// TIA Portal V17 export
// export: Created 2022-07-20T07:01:34.0811229Z, ExportSetting WithDefaults, DisplayName Totally Integrated Automation Portal, DisplayVersion V17, DisplayName TIA Portal Openness, DisplayVersion V17, DisplayName TIA Portal Version Control Interface, DisplayVersion V17, DisplayName SINAMICS Startdrive Advanced, DisplayVersion V17, DisplayName SINAMICS Startdrive G130, G150, S120, S150, SINAMICS MV, S210, DisplayVersion V17, DisplayName SINAMICS Startdrive G110M, G120, G120C, G120D, G120P, G115D, DisplayVersion V17, DisplayName STEP 7 Professional, DisplayVersion V17, DisplayName STEP 7 Safety, DisplayVersion V17, DisplayName WinCC Advanced, DisplayVersion V17
FUNCTION_BLOCK "FB10324_PrinterCompactCapingStation"   // FB10324, LAD
{ S7_Optimized_Access := 'TRUE' }
VERSION : 0.1
// stored: AutoNumber false, IsIECCheckEnabled false, IsRetainMemResEnabled false, MemoryReserve 100, SetENOAutomatically false, UDAEnableTagReadback false
   VAR_OUTPUT
      CapingStation_FillingDone : Bool;
      CapingStationLongOverflowingDone : Bool;
      CapingStationShortOverflowingDone : Bool;
      CapingStationEmptyingDone : Bool;
      CapingStation_WashupSolenoidValve_1_2 : Bool;
      CapingStation_WashupSolenoidValve_3_4 : Bool;
      CapingStation_EmptyingSolenoidValve_1_2 : Bool;
      CapingStation_EmptyingSolenoidValve_3_4 : Bool;
      CapingStation_CleaningSolenoidValve_1_2 : Bool;
      CapingStation_CleaningSolenoidValve_3_4 : Bool;
      CapingStation_WashupPump : Bool;
      CapingStation_EmptyingPump : Bool;
   END_VAR
   VAR_IN_OUT
      RequestFillingCapingStation : Bool;
      RequestLongOverflowingCapingStation : Bool;
      RequestShortOverflowingCapingStation : Bool;
      RequestEmptyingCapingStation : Bool;
   END_VAR
   VAR
      ManagerCapingStationStateDiagram : Int;
      TON_FillingCapingStation : TON_TIME;
      TON_LongOverflowingCapingStation : TON_TIME;
      TON_ShortOverflowingCapingStation : TON_TIME;
      TON_EmptyingCapingStation : TON_TIME;
      R_TRIG_RequestFillingCapingStation { S7_SetPoint := 'True'} : R_TRIG;
      R_TRIG_RequestLongOverflowingCapingStation { S7_SetPoint := 'True'} : R_TRIG;
      R_TRIG_RequestShortOverflowingCapingStation { S7_SetPoint := 'True'} : R_TRIG;
      R_TRIG_RequestEmptyingCapingStation { S7_SetPoint := 'True'} : R_TRIG;
   END_VAR
   VAR CONSTANT
      "0_WAIT_FOR_REQUEST_CAPING_STATION" : Int;
      "10_REQUEST_FILING_CAPING_STATION" : Int := 10;
      "20_REQUEST_LONG_OVERFLOWING_CAPING_STATION" : Int := 20;
      "30_REQUEST_SHORT_OVERFLOWING_CAPING_STATION" : Int := 30;
      "40_REQUEST_EMPTYING_CAPING_STATION" : Int := 40;
      "10000_ALL_ACTIONS_DONE" : Int := 10000;
   END_VAR
BEGIN

REGION Network 1 (SCL): FirstScan
   IF "FirstScan" THEN
       ;
   END_IF;
END_REGION

REGION Network 2 (SCL): Edge Signals & Timers
   REGION EDGE SIGNAL

       #R_TRIG_RequestFillingCapingStation(CLK := #RequestFillingCapingStation);
       #R_TRIG_RequestLongOverflowingCapingStation(CLK := #RequestLongOverflowingCapingStation);
       #R_TRIG_RequestShortOverflowingCapingStation(CLK := #RequestShortOverflowingCapingStation);
       #R_TRIG_RequestEmptyingCapingStation(CLK := #RequestEmptyingCapingStation);

   END_REGION

   REGION

       #TON_FillingCapingStation(IN := #ManagerCapingStationStateDiagram = #"10_REQUEST_FILING_CAPING_STATION",
                                 PT := T#27s);
       #TON_LongOverflowingCapingStation(IN := #ManagerCapingStationStateDiagram = #"20_REQUEST_LONG_OVERFLOWING_CAPING_STATION",
                                         PT := T#5s);
       #TON_ShortOverflowingCapingStation(IN := #ManagerCapingStationStateDiagram = #"30_REQUEST_SHORT_OVERFLOWING_CAPING_STATION",
                                          PT := T#2s);
       #TON_EmptyingCapingStation(IN := #ManagerCapingStationStateDiagram = #"40_REQUEST_EMPTYING_CAPING_STATION",
                                  PT := T#30s);

   END_REGION
END_REGION

REGION Network 3 (SCL): Caping Station Statement Management
END_REGION

REGION Network 4 (SCL): Caping Station Management
   CASE #ManagerCapingStationStateDiagram OF

       #"0_WAIT_FOR_REQUEST_CAPING_STATION" :
           IF #R_TRIG_RequestFillingCapingStation.Q AND NOT (#CapingStation_FillingDone) THEN
               #ManagerCapingStationStateDiagram := #"10_REQUEST_FILING_CAPING_STATION";
           ELSIF #CapingStation_FillingDone AND #R_TRIG_RequestLongOverflowingCapingStation.Q THEN
               #ManagerCapingStationStateDiagram := #"20_REQUEST_LONG_OVERFLOWING_CAPING_STATION";
           ELSIF #CapingStation_FillingDone AND #R_TRIG_RequestShortOverflowingCapingStation.Q THEN
               #ManagerCapingStationStateDiagram := #"30_REQUEST_SHORT_OVERFLOWING_CAPING_STATION";
           ELSIF #R_TRIG_RequestEmptyingCapingStation.Q THEN
               #ManagerCapingStationStateDiagram := #"40_REQUEST_EMPTYING_CAPING_STATION";
           END_IF;

       #"10_REQUEST_FILING_CAPING_STATION" :
           #CapingStation_WashupPump := TRUE;
           #CapingStation_WashupSolenoidValve_1_2 := TRUE;
           #CapingStation_WashupSolenoidValve_3_4 := TRUE;
           #CapingStation_CleaningSolenoidValve_1_2 := TRUE;
           #CapingStation_CleaningSolenoidValve_3_4 := TRUE;
           IF #TON_FillingCapingStation.Q THEN
               #RequestFillingCapingStation := FALSE;
               #CapingStation_FillingDone := TRUE;
               #CapingStation_WashupPump := FALSE;
               #CapingStation_WashupSolenoidValve_1_2 := FALSE;
               #CapingStation_WashupSolenoidValve_3_4 := FALSE;
               #CapingStation_CleaningSolenoidValve_1_2 := FALSE;
               #CapingStation_CleaningSolenoidValve_3_4 := FALSE;
               #ManagerCapingStationStateDiagram := #"10000_ALL_ACTIONS_DONE";
           END_IF;

       #"20_REQUEST_LONG_OVERFLOWING_CAPING_STATION" :
           #CapingStation_WashupPump := TRUE;
           #CapingStation_WashupSolenoidValve_1_2 := TRUE;
           #CapingStation_WashupSolenoidValve_3_4 := TRUE;
           #CapingStation_CleaningSolenoidValve_1_2 := TRUE;
           #CapingStation_CleaningSolenoidValve_3_4 := TRUE;
           IF #TON_LongOverflowingCapingStation.Q THEN
               #RequestLongOverflowingCapingStation := FALSE;
               #CapingStationLongOverflowingDone := TRUE;
               #CapingStation_WashupPump := FALSE;
               #CapingStation_WashupSolenoidValve_1_2 := FALSE;
               #CapingStation_WashupSolenoidValve_3_4 := FALSE;
               #CapingStation_CleaningSolenoidValve_1_2 := FALSE;
               #CapingStation_CleaningSolenoidValve_3_4 := FALSE;
               #ManagerCapingStationStateDiagram := #"10000_ALL_ACTIONS_DONE";
           END_IF;

       #"30_REQUEST_SHORT_OVERFLOWING_CAPING_STATION" :
           #CapingStation_WashupPump := TRUE;
           #CapingStation_WashupSolenoidValve_1_2 := TRUE;
           #CapingStation_WashupSolenoidValve_3_4 := TRUE;
           #CapingStation_CleaningSolenoidValve_1_2 := TRUE;
           #CapingStation_CleaningSolenoidValve_3_4 := TRUE;
           IF #TON_ShortOverflowingCapingStation.Q THEN
               #RequestShortOverflowingCapingStation := FALSE;
               #CapingStationShortOverflowingDone := TRUE;
               #CapingStation_WashupPump := FALSE;
               #CapingStation_WashupSolenoidValve_1_2 := FALSE;
               #CapingStation_WashupSolenoidValve_3_4 := FALSE;
               #CapingStation_CleaningSolenoidValve_1_2 := FALSE;
               #CapingStation_CleaningSolenoidValve_3_4 := FALSE;
               #ManagerCapingStationStateDiagram := #"10000_ALL_ACTIONS_DONE";
           END_IF;

       #"40_REQUEST_EMPTYING_CAPING_STATION" :
           #CapingStation_EmptyingPump:= TRUE;
           #CapingStation_EmptyingSolenoidValve_1_2 := TRUE;
           #CapingStation_EmptyingSolenoidValve_3_4 := TRUE;
           IF #TON_EmptyingCapingStation.Q THEN
               #CapingStationEmptyingDone := TRUE;
               #RequestEmptyingCapingStation := FALSE;
               #CapingStation_FillingDone := FALSE;
               #CapingStation_EmptyingPump := FALSE;
               #CapingStation_EmptyingSolenoidValve_1_2 := FALSE;
               #CapingStation_EmptyingSolenoidValve_3_4 := FALSE;
               #ManagerCapingStationStateDiagram := #"10000_ALL_ACTIONS_DONE";
           END_IF;

       #"10000_ALL_ACTIONS_DONE" :
           #CapingStation_WashupPump := FALSE;
           #CapingStation_EmptyingPump := FALSE;
           #CapingStation_WashupSolenoidValve_1_2 := FALSE;
           #CapingStation_WashupSolenoidValve_3_4 := FALSE;
           #CapingStation_CleaningSolenoidValve_1_2 := FALSE;
           #CapingStation_CleaningSolenoidValve_3_4 := FALSE;
           #CapingStation_EmptyingSolenoidValve_1_2 := FALSE;
           #CapingStation_EmptyingSolenoidValve_3_4 := FALSE;
           #CapingStationShortOverflowingDone := FALSE;
           #CapingStationLongOverflowingDone := FALSE;
           #CapingStationEmptyingDone := FALSE;
           #ManagerCapingStationStateDiagram := #"0_WAIT_FOR_REQUEST_CAPING_STATION";


   END_CASE;
END_REGION

REGION Network 5 (SCL): Caping Station State Management
END_REGION
END_FUNCTION_BLOCK
